(* IEC 61131-3 sources: PTConstructor/Examples, 13 files *)

(* ---- AutoCarWash.st ---- *)
PROGRAM AutoCarWash
  VAR_INPUT
    Master_Start : BOOL := false;
    Car_Detection : BOOL := false;
    Limit_Switch : BOOL := false;
    Master_Stop : BOOL := false;
  END_VAR
  VAR_OUTPUT
    Master_Coil : BOOL := false;
    Soap_Sprinkler : BOOL := false;
    Washer : BOOL := false;
    Conveyor : BOOL := false;
    Dryer : BOOL := false;
  END_VAR
  VAR
    SoapingTimeDN : BOOL := false;
    WashingTimeDN : BOOL := false;
    DryingTimeDN : BOOL := false;
    SoapingTime : TON;
    WashingTime : TON;
    DryingTime : TON;
  END_VAR

  Master_Coil := NOT(Master_Stop) AND (Master_Coil OR Master_Start);
  Soap_Sprinkler := NOT(SoapingTimeDN) AND Car_Detection AND Master_Coil;
  SoapingTime(IN := Car_Detection AND Master_Coil, PT := T#200ms);
  SoapingTimeDN := SoapingTime.Q;
  Washer := NOT(WashingTimeDN) AND SoapingTimeDN AND Master_Coil;
  WashingTime(IN := (Dryer OR SoapingTimeDN) AND Master_Coil, PT := T#250ms);
  WashingTimeDN := WashingTime.Q;
  Conveyor := NOT(Limit_Switch) AND WashingTimeDN AND Master_Coil;
  Dryer := NOT(DryingTimeDN) AND WashingTimeDN AND Master_Coil;
  DryingTime(IN := (Dryer OR WashingTimeDN) AND Master_Coil, PT := T#100ms);
  DryingTimeDN := DryingTime.Q;
END_PROGRAM

CONFIGURATION Config0

  RESOURCE Res0 ON PLC
    TASK task0(INTERVAL := T#20ms,PRIORITY := 0);
    PROGRAM instance0 WITH task0 : AutoCarWash;
  END_RESOURCE
END_CONFIGURATION

(* ---- BottleFillingSystem.st ---- *)
PROGRAM BottleFillingSystem
  VAR_INPUT
    Start : BOOL;
    Stop : BOOL;
  END_VAR
  VAR_OUTPUT
    MasterCoil : BOOL;
  END_VAR
  VAR_INPUT
    Input : UDINT;
  END_VAR
  VAR
    DivResult : UDINT;
    MulResult : UDINT;
  END_VAR
  VAR_OUTPUT
    IPConverter : UDINT;
  END_VAR
  VAR
    DIV9_ENO : BOOL;
    DIV9_OUT : UDINT;
    MUL15_ENO : BOOL;
    MUL15_OUT : UDINT;
    MOVE21_ENO : BOOL;
    MOVE21_OUT : UDINT;
  END_VAR

  MasterCoil := NOT(Stop) AND (MasterCoil OR Start);
  DIV9_OUT := DIV(EN := MasterCoil, IN1 := Input, IN2 := 1000, ENO => DIV9_ENO);
  IF DIV9_ENO THEN
      DivResult := DIV9_OUT;
  END_IF;
  MUL15_OUT := MUL(EN := MasterCoil, IN1 := DivResult, IN2 := 902, ENO => MUL15_ENO);
  IF MUL15_ENO THEN
      MulResult := MUL15_OUT;
  END_IF;
  MOVE21_OUT := MOVE(EN := MasterCoil, IN := MulResult, ENO => MOVE21_ENO);
  IF MOVE21_ENO THEN
      IPConverter := MOVE21_OUT;
  END_IF;
END_PROGRAM

CONFIGURATION Config0

  RESOURCE Res0 ON PLC
    TASK task0(INTERVAL := T#20ms,PRIORITY := 0);
    PROGRAM instance0 WITH task0 : BottleFillingSystem;
  END_RESOURCE
END_CONFIGURATION

(* ---- BurnedChipsRemove.st ---- *)
PROGRAM BurnedChipsRemove
  VAR_INPUT
    Start : BOOL := false;
    Stop : BOOL := false;
  END_VAR
  VAR_OUTPUT
    MasterCoil : BOOL := false;
    Conveyor : BOOL := false;
    LightSource : BOOL := false;
  END_VAR
  VAR_INPUT
    LightDependentResistors1 : BOOL;
    LightDependentResistors2 : BOOL;
  END_VAR
  VAR
    BitLatching1 : BOOL;
    BitLatching2 : BOOL;
  END_VAR
  VAR_OUTPUT
    Blowers1 : BOOL;
    Blowers2 : BOOL;
  END_VAR
  VAR
    TimerToActivateBlowerDN : BOOL := false;
    TimerToActivateBlower : TON;
  END_VAR

  MasterCoil := NOT(Stop) AND (MasterCoil OR Start);
  Conveyor := MasterCoil;
  LightSource := MasterCoil;
  BitLatching1 := NOT(TimerToActivateBlowerDN) AND (BitLatching1 OR LightDependentResistors1);
  BitLatching2 := NOT(TimerToActivateBlowerDN) AND (BitLatching2 OR LightDependentResistors2);
  TimerToActivateBlower(IN := (BitLatching1 OR BitLatching2) AND MasterCoil, PT := T#10ms);
  TimerToActivateBlowerDN := TimerToActivateBlower.Q;
  Blowers1 := TimerToActivateBlowerDN AND BitLatching1 AND MasterCoil;
  Blowers2 := TimerToActivateBlowerDN AND BitLatching2 AND MasterCoil;
END_PROGRAM

CONFIGURATION Config0

  RESOURCE Res0 ON PLC
    TASK task0(INTERVAL := T#20ms,PRIORITY := 0);
    PROGRAM instance0 WITH task0 : BurnedChipsRemove;
  END_RESOURCE
END_CONFIGURATION

(* ---- CleaningRinsingBottles.st ---- *)
PROGRAM CleaningRinsingBottles
  VAR_INPUT
    Start : BOOL := false;
    Stop : BOOL := false;
    BottleEnter : BOOL := false;
    BottleLeave : BOOL := false;
    UpsideDown : BOOL := false;
  END_VAR
  VAR_OUTPUT
    MasterCoil : BOOL := false;
    ClipHold : BOOL := false;
    TurnBottleForward : BOOL := false;
    TurnBottleReverse : BOOL := false;
    WaterSupply : BOOL := false;
    ClipRelease : BOOL := false;
  END_VAR
  VAR
    TurnBottleTimeDN : BOOL := false;
    SprinkleWaterTimeDN : BOOL := false;
    LeaveBottleTimeDN : BOOL := false;
    TurnBottleTime : TON;
    SprinkleWaterTime : TON;
    LeaveBottleTime : TON;
  END_VAR

  MasterCoil := NOT(Stop) AND (MasterCoil OR Start);
  ClipHold := NOT(BottleLeave) AND (BottleEnter OR ClipHold) AND MasterCoil;
  TurnBottleTime(IN := ClipHold AND MasterCoil, PT := T#2000ms);
  TurnBottleTimeDN := TurnBottleTime.Q;
  TurnBottleForward := TurnBottleTimeDN AND MasterCoil;
  WaterSupply := NOT(SprinkleWaterTimeDN) AND (UpsideDown OR WaterSupply) AND TurnBottleForward AND MasterCoil;
  SprinkleWaterTime(IN := WaterSupply AND MasterCoil, PT := T#2000ms);
  SprinkleWaterTimeDN := SprinkleWaterTime.Q;
  TurnBottleReverse := NOT(BottleEnter) AND (BottleLeave OR TurnBottleReverse) AND MasterCoil;
  LeaveBottleTime(IN := TurnBottleReverse AND MasterCoil, PT := T#3000ms);
  LeaveBottleTimeDN := LeaveBottleTime.Q;
  ClipRelease := NOT(BottleEnter) AND LeaveBottleTimeDN AND MasterCoil;
END_PROGRAM

CONFIGURATION Config0

  RESOURCE Res0 ON PLC
    TASK task0(INTERVAL := T#20ms,PRIORITY := 0);
    PROGRAM instance0 WITH task0 : CleaningRinsingBottles;
  END_RESOURCE
END_CONFIGURATION

(* ---- ControlSprayPainting.st ---- *)
PROGRAM ControlSprayPainting
  VAR_INPUT
    Start : BOOL := false;
    Stop : BOOL := false;
    Hanger : BOOL := false;
    PartDetection : BOOL := false;
  END_VAR
  VAR_OUTPUT
    MasterCoil : BOOL := false;
    Oven : BOOL := false;
    Spray : BOOL := false;
  END_VAR
  VAR
    BitShift : BYTE := 0;
    AND17_ENO : BOOL;
    AND17_OUT : BYTE;
    SHL13_ENO : BOOL;
    SHL13_OUT : BYTE;
    AND26_OUT : BYTE;
    GT28_OUT : BOOL;
  END_VAR

  MasterCoil := NOT(Stop) AND (MasterCoil OR Start);
  Oven := MasterCoil;
  AND17_OUT := AND(EN := PartDetection, IN1 := BitShift, IN2 := 1, ENO => AND17_ENO);
  IF AND17_ENO THEN
      BitShift := AND17_OUT;
  END_IF;
  SHL13_OUT := SHL(EN := Hanger, IN := BitShift, N := 1, ENO => SHL13_ENO);
  IF SHL13_ENO THEN
      BitShift := SHL13_OUT;
  END_IF;
  AND26_OUT := AND(BitShift, 4);
  GT28_OUT := GT(AND26_OUT, 0);
  Spray := GT28_OUT;
END_PROGRAM

CONFIGURATION Config0

  RESOURCE Res0 ON PLC
    TASK task0(INTERVAL := T#20ms,PRIORITY := 0);
    PROGRAM instance0 WITH task0 : ControlSprayPainting;
  END_RESOURCE
END_CONFIGURATION

(* ---- CountPackParts.st ---- *)
PROGRAM CountPackParts
  VAR_INPUT
    Start : BOOL := false;
    Stop : BOOL := false;
    PartDetection : BOOL := false;
    BoxDetection : BOOL := false;
  END_VAR
  VAR_OUTPUT
    LatchingBit : BOOL := false;
    LatchingMotor : BOOL := false;
    ConveyorBelt1 : BOOL := false;
    ConveyorBelt2 : BOOL := false;
  END_VAR
  VAR
    StopConveyorTimeDN : BOOL := false;
    PartCounterDN : BOOL := false;
    PartCounter : CTU;
    StopConveyorTime : TON;
    R_TRIG1 : R_TRIG;
  END_VAR

  LatchingBit := NOT(Stop) AND (LatchingBit OR Start);
  ConveyorBelt1 := NOT(StopConveyorTimeDN) AND (BoxDetection OR ConveyorBelt1) AND LatchingBit;
  R_TRIG1(CLK := PartDetection AND LatchingBit);
  PartCounter(CU := R_TRIG1.Q, R := PartCounterDN, PV := 5);
  PartCounterDN := PartCounter.Q;
  StopConveyorTime(IN := LatchingMotor AND LatchingBit, PT := T#2000ms);
  StopConveyorTimeDN := StopConveyorTime.Q;
  LatchingMotor := NOT(StopConveyorTimeDN) AND (LatchingMotor OR PartCounterDN) AND LatchingBit;
  ConveyorBelt2 := NOT(BoxDetection) AND (ConveyorBelt2 OR PartCounterDN) AND LatchingBit;
END_PROGRAM

CONFIGURATION Config0

  RESOURCE Res0 ON PLC
    TASK task0(INTERVAL := T#20ms,PRIORITY := 0);
    PROGRAM instance0 WITH task0 : CountPackParts;
  END_RESOURCE
END_CONFIGURATION

(* ---- DrillingParts.st ---- *)
PROGRAM DrillingParts
  VAR_INPUT
    Start : BOOL := false;
    Stop : BOOL := false;
  END_VAR
  VAR_OUTPUT
    MasterCoil : BOOL := false;
    ClampingDevice : BOOL := false;
    DrillingMotor : BOOL := false;
    MotorDown : BOOL := false;
    MotorUp : BOOL := false;
  END_VAR
  VAR_INPUT
    ObjectDetector : BOOL := false;
    LowerLimit : BOOL := false;
    UpperLimit : BOOL := false;
  END_VAR

  MasterCoil := NOT(Stop) AND (MasterCoil OR Start);
  ClampingDevice := NOT(LowerLimit) AND (NOT(UpperLimit) OR ObjectDetector) AND (DrillingMotor OR ObjectDetector) AND MasterCoil;
  DrillingMotor := (NOT(UpperLimit) OR ObjectDetector) AND (DrillingMotor OR ObjectDetector) AND MasterCoil;
  MotorDown := NOT(LowerLimit) AND (NOT(UpperLimit) OR ObjectDetector) AND (DrillingMotor OR ObjectDetector) AND MasterCoil;
  MotorUp := NOT(UpperLimit) AND (LowerLimit OR MotorUp) AND MasterCoil;
END_PROGRAM

CONFIGURATION Config0

  RESOURCE Res0 ON PLC
    TASK task0(INTERVAL := T#20ms,PRIORITY := 0);
    PROGRAM instance0 WITH task0 : DrillingParts;
  END_RESOURCE
END_CONFIGURATION

(* ---- JumpToOtherProc.st ---- *)
PROGRAM JumpToOtherProc
  VAR_INPUT
    JumpLabel : BOOL := false;
    A : BOOL := false;
    B : BOOL := false;
    C : BOOL := false;
    Sensor : BOOL := false;
  END_VAR
  VAR_OUTPUT
    O0 : BOOL := false;
    O1 : BOOL := false;
    O2 : BOOL := false;
    O3 : BOOL := false;
  END_VAR
  VAR_IN_OUT
    Jump : BOOL;
  END_VAR

  Jump := JumpLabel;
  O0 := A;
  O1 := B;
  O2 := C;
  O3 := Sensor AND Jump;
END_PROGRAM

CONFIGURATION Config0

  RESOURCE Res0 ON PLC
    TASK task0(INTERVAL := T#20ms,PRIORITY := 0);
    PROGRAM instance0 WITH task0 : JumpToOtherProc;
  END_RESOURCE
END_CONFIGURATION

(* ---- MathFuncs.st ---- *)
PROGRAM MathFuncs
  VAR_INPUT
    InputToAdd : BOOL;
    InputToSub : BOOL;
    InputToMul : BOOL;
    InputToDiv : BOOL;
    InputToSqrt : BOOL;
    InputToNeg : BOOL;
    InputNum0 : DINT;
    InputNum1 : DINT;
    InputNum2 : DINT;
    InputNum3 : DINT;
    InputNum4 : DINT;
    InputNum5 : DINT;
    InputNum6 : DINT;
    InputNum7 : DINT;
    InputNum8 : REAL;
  END_VAR
  VAR_OUTPUT
    Output0 : DINT;
    Output1 : REAL;
  END_VAR
  VAR
    ADD3_ENO : BOOL;
    ADD3_OUT : DINT;
    SUB10_ENO : BOOL;
    SUB10_OUT : DINT;
    MUL17_ENO : BOOL;
    MUL17_OUT : DINT;
    DIV24_ENO : BOOL;
    DIV24_OUT : DINT;
    SQRT31_ENO : BOOL;
    SQRT31_OUT : REAL;
  END_VAR

  ADD3_OUT := ADD(EN := InputToAdd, IN1 := InputNum0, IN2 := InputNum1, ENO => ADD3_ENO);
  IF ADD3_ENO THEN
      Output0 := ADD3_OUT;
  END_IF;
  SUB10_OUT := SUB(EN := InputToSub, IN1 := InputNum2, IN2 := InputNum3, ENO => SUB10_ENO);
  IF SUB10_ENO THEN
      Output0 := SUB10_OUT;
  END_IF;
  MUL17_OUT := MUL(EN := InputToMul, IN1 := InputNum4, IN2 := InputNum5, ENO => MUL17_ENO);
  IF MUL17_ENO THEN
      Output0 := MUL17_OUT;
  END_IF;
  DIV24_OUT := DIV(EN := InputToDiv, IN1 := InputNum6, IN2 := InputNum7, ENO => DIV24_ENO);
  IF DIV24_ENO THEN
      Output0 := DIV24_OUT;
  END_IF;
  SQRT31_OUT := SQRT(EN := InputToSqrt, IN := InputNum8, ENO => SQRT31_ENO);
  IF SQRT31_ENO THEN
      Output1 := SQRT31_OUT;
  END_IF;
END_PROGRAM

CONFIGURATION Config0

  RESOURCE Res0 ON PLC
    TASK task0(INTERVAL := T#20ms,PRIORITY := 0);
    PROGRAM instance0 WITH task0 : MathFuncs;
  END_RESOURCE
END_CONFIGURATION

(* ---- MixingDevice.st ---- *)
PROGRAM MixingDevice
  VAR_INPUT
    Start : BOOL := false;
    Stop : BOOL := false;
  END_VAR
  VAR_OUTPUT
    MasterCoil : BOOL := false;
  END_VAR
  VAR_INPUT
    MaterialA : BOOL := false;
    MaterialB : BOOL := false;
    LowLevel : BOOL := false;
  END_VAR
  VAR_OUTPUT
    InletValveA : BOOL := false;
    InletValveB : BOOL := false;
    AgitatorMotor : BOOL := false;
    OutletValve : BOOL := false;
  END_VAR
  VAR
    TimerMixDN : BOOL := false;
    TimerMix : TON;
  END_VAR

  MasterCoil := NOT(Stop) AND (MasterCoil OR Start);
  InletValveA := NOT(MaterialA) AND (InletValveA OR LowLevel OR Start) AND MasterCoil;
  InletValveB := NOT(MaterialB) AND (InletValveB OR MaterialA) AND MasterCoil;
  AgitatorMotor := NOT(TimerMixDN) AND (AgitatorMotor OR MaterialB) AND MasterCoil;
  TimerMix(IN := AgitatorMotor AND MasterCoil, PT := T#200ms);
  TimerMixDN := TimerMix.Q;
  OutletValve := NOT(LowLevel) AND TimerMixDN AND MasterCoil;
END_PROGRAM

CONFIGURATION Config0

  RESOURCE Res0 ON PLC
    TASK task0(INTERVAL := T#20ms,PRIORITY := 0);
    PROGRAM instance0 WITH task0 : MixingDevice;
  END_RESOURCE
END_CONFIGURATION

(* ---- MotorForwardBackward.st ---- *)
PROGRAM MotorFB
  VAR_INPUT
    ForwardStart : BOOL := false;
    ReverseStart : BOOL := false;
    Stop : BOOL := false;
  END_VAR
  VAR_OUTPUT
    LatchedF : BOOL := false;
    ForwardContactor : BOOL := false;
    LatchedR : BOOL := false;
    ReverseContactor : BOOL := false;
  END_VAR
  VAR
    DelayFDN : BOOL := false;
    DelayRDN : BOOL := false;
    DelayF : TOF;
    DelayR : TOF;
  END_VAR

  LatchedF := ForwardStart AND ForwardStart AND NOT(Stop) OR NOT(LatchedR) AND (ForwardStart OR LatchedF) AND NOT(Stop);
  ForwardContactor := NOT(DelayFDN) AND LatchedF;
  DelayF(IN := LatchedF, PT := T#120ms);
  DelayFDN := DelayF.Q;
  LatchedR := NOT(LatchedF) AND (LatchedR OR ReverseStart) AND NOT(Stop) OR ReverseStart AND ReverseStart AND NOT(Stop);
  ReverseContactor := NOT(DelayRDN) AND LatchedR;
  DelayR(IN := LatchedR, PT := T#120ms);
  DelayRDN := DelayR.Q;
END_PROGRAM

CONFIGURATION Config0

  RESOURCE Res0 ON PLC
    TASK task0(INTERVAL := T#20ms,PRIORITY := 0);
    PROGRAM instance0 WITH task0 : MotorFB;
  END_RESOURCE
END_CONFIGURATION

(* ---- QualityControl.st ---- *)
PROGRAM QualityControl
  VAR_INPUT
    Start : BOOL;
    Stop : BOOL;
    Detector : BOOL;
  END_VAR
  VAR
    LatchingCoil : BOOL;
  END_VAR
  VAR_OUTPUT
    ConveyorMotors : BOOL;
    OperateGate : BOOL;
  END_VAR
  VAR
    CounterDN : BOOL;
    TimerDN : BOOL;
    Counter : CTU;
    Timer : TON;
    R_TRIG1 : R_TRIG;
  END_VAR

  LatchingCoil := NOT(Stop) AND (LatchingCoil OR Start);
  ConveyorMotors := LatchingCoil;
  R_TRIG1(CLK := Detector AND LatchingCoil);
  Counter(CU := R_TRIG1.Q, R := TimerDN, PV := 1000);
  CounterDN := Counter.Q;
  OperateGate := CounterDN AND LatchingCoil;
  Timer(IN := CounterDN AND LatchingCoil, PT := T#20ms);
  TimerDN := Timer.Q;
END_PROGRAM

CONFIGURATION Config0

  RESOURCE Res0 ON PLC
    TASK task0(INTERVAL := T#20ms,PRIORITY := 0);
    PROGRAM instance0 WITH task0 : QualityControl;
  END_RESOURCE
END_CONFIGURATION

(* ---- SeparateParts.st ---- *)
PROGRAM SeparateParts
  VAR_INPUT
    Start : BOOL := False;
    Stop : BOOL := False;
  END_VAR
  VAR_OUTPUT
    MasterCoil : BOOL := False;
  END_VAR
  VAR_INPUT
    DetectBigParts : BOOL := False;
  END_VAR
  VAR_OUTPUT
    GateSolenoidCoil : BOOL := False;
    TimerGateDN : BOOL := False;
  END_VAR
  VAR
    TimerGate : TON;
  END_VAR

  MasterCoil := NOT(Stop) AND (MasterCoil OR Start);
  GateSolenoidCoil := NOT(TimerGateDN) AND (DetectBigParts OR GateSolenoidCoil) AND MasterCoil;
  TimerGate(IN := GateSolenoidCoil AND MasterCoil, PT := T#20ms);
  TimerGateDN := TimerGate.Q;
END_PROGRAM

CONFIGURATION Config0

  RESOURCE Res0 ON PLC
    TASK task0(INTERVAL := T#20ms,PRIORITY := 0);
    PROGRAM instance0 WITH task0 : SeparateParts;
  END_RESOURCE
END_CONFIGURATION
